KUKA KRL program: braketestselftest.src, braketestselftest.dat

--- braketestselftest.src ---
&ACCESS RVP
&REL 1
&PARAM TEMPLATE = C:\KRC\Roboter\Template\ExpertVorgabe
&PARAM EDITMASK = *
DEF BrakeTestSelfTest( )
;FOLD perform brake test self test

;ENDFOLD
;FOLD ;%{H}
BrakeTestReq(TRUE)
;ENDFOLD
END

--- braketestselftest.dat ---
&ACCESS RVP
&REL 1
&PARAM TEMPLATE = C:\KRC\Roboter\Template\ExpertVorgabe
&PARAM EDITMASK = *
DEFDAT braketestselftest PUBLIC

ENDDAT
